// TwinCAT 3 PLC project PLC1
// ProgramVersion: 3.1.4023.0
// libraries:
//   Tc2_Standard, * (Beckhoff Automation GmbH)
//   Tc2_System, * (Beckhoff Automation GmbH)
//   Tc3_Module, * (Beckhoff Automation GmbH)
// project tree:
//   DUTs/ udtLogging.TcDUT, udtZoneManager.TcDUT
//   GVLs/ DataProces2.TcGVL, DataConfig.TcGVL, GVLDataproces.TcGVL, GVLtest1.TcGVL, GVLtest10.TcGVL, GVLtest2.TcGVL
//   / PlcTask.TcTTO
//   POUs/ fb_motor.TcPOU, fb_motor_1.TcPOU, fb_motor_2.TcPOU, MAIN.TcPOU
// real-time tasks:
//   TASK PlcTask: cycle T#10ms, priority 20, ADS port 350
// I/O:
//   DEVICE Device 1 (EtherCAT), AmsNetId 192.168.153.1.2.1
//     Term 1 (EK1200) [EK1200-5000 EtherCAT Power supply (2A E-Bus)]
//       Term 4 (EL1008)
//       Term 5 (EL1008) [EL1008 8Ch. Dig. Input 24V, 3ms]
//       Term 6 (EL1008) [EL1008 8Ch. Dig. Input 24V, 3ms]
//       Term 7 (EL1008) [EL1008 8Ch. Dig. Input 24V, 3ms]
//       Term 8 (EL1008) [EL1008 8Ch. Dig. Input 24V, 3ms]
//       Term 9 (EL1008) [EL1008 8Ch. Dig. Input 24V, 3ms]
//       Term 10 (EL1008) [EL1008 8Ch. Dig. Input 24V, 3ms]
//       Term 11 (EL1008) [EL1008 8Ch. Dig. Input 24V, 3ms]
//       Term 2 (EL1008) [EL1008 8Ch. Dig. Input 24V, 3ms]
//       Term 13 (EL2008) [EL2008 8Ch. Dig. Output 24V, 0.5A]
//       Term 14 (EL2008) [EL2008 8Ch. Dig. Output 24V, 0.5A]
//       Term 15 (EL2008) [EL2008 8Ch. Dig. Output 24V, 0.5A]
//       Term 16 (EL2008) [EL2008 8Ch. Dig. Output 24V, 0.5A]
//       Term 12 (EL2008) [EL2008 8Ch. Dig. Output 24V, 0.5A]
//       Term 3 (EL9011)

CONFIGURATION PLC1
    RESOURCE PLC ON TwinCAT3
        TASK PlcTask(INTERVAL := T#10ms, PRIORITY := 20);
        PROGRAM MAIN WITH PlcTask : MAIN;
    END_RESOURCE
END_CONFIGURATION

// ---- DUTs/udtLogging.TcDUT
TYPE udtLogging :
STRUCT
	StartLog	:	BOOL;
	LogID		:	INT;
END_STRUCT
END_TYPE

// ---- DUTs/udtZoneManager.TcDUT
TYPE udtZoneManager :
STRUCT
	Auto	:	BOOL;
	Manual	:	BOOL;
	Start	:	BOOL;
	Stop	:	BOOL;
END_STRUCT
END_TYPE

// ---- GVLs/DataProces2.TcGVL
{attribute 'qualified_only'}
VAR_GLOBAL
	test: BOOL;
END_VAR

// ---- GVLs/DataConfig.TcGVL
{attribute 'qualified_only'}
VAR_GLOBAL
	test: BOOL;
END_VAR

// ---- GVLs/GVLDataproces.TcGVL
{attribute 'qualified_only'}
VAR_GLOBAL
	Test :BOOL;
	Data :ARRAY[0..100] OF INT;
	DAtatekst : STRING[255];
	extraData : BOOL;
END_VAR

// ---- GVLs/GVLtest1.TcGVL
{attribute 'qualified_only'}
VAR_GLOBAL
	test1: BOOL;
END_VAR

// ---- GVLs/GVLtest10.TcGVL
{attribute 'qualified_only'}
VAR_GLOBAL
END_VAR

// ---- GVLs/GVLtest2.TcGVL
{attribute 'qualified_only'}
VAR_GLOBAL
	truefalse	:	BOOL;
END_VAR

// ---- POUs/MAIN.TcPOU
PROGRAM MAIN
VAR
	fbMotor1: fb_motor;
	fbmotor2: fb_motor;
END_VAR


fbMotor1(bStart:= true, bStop:= true, bStatus=> );

END_PROGRAM

// ---- POUs/fb_motor.TcPOU
FUNCTION_BLOCK fb_motor
VAR_INPUT
	bStart, bStop : BOOL;
	
END_VAR
VAR_OUTPUT
	bStatus : BOOL;
END_VAR
VAR
END_VAR

END_FUNCTION_BLOCK

// ---- POUs/fb_motor_1.TcPOU
FUNCTION_BLOCK fb_motor_1
VAR_INPUT
	bStart, bStop : BOOL;
	
END_VAR
VAR_OUTPUT
	bStatus : BOOL;
END_VAR
VAR
END_VAR

END_FUNCTION_BLOCK

// ---- POUs/fb_motor_2.TcPOU
FUNCTION_BLOCK fb_motor_2
VAR_INPUT
	bStart, bStop : BOOL;
	
END_VAR
VAR_OUTPUT
	bStatus : BOOL;
END_VAR
VAR
END_VAR

END_FUNCTION_BLOCK
